// SIMATIC S7-200 project (STEP 7-Micro/WIN), CPU 221 REL 01.10

SYMBOL_TABLE USER1
bezczynnosc_do_za_gorac M1.7     // w彻cz wiatrak
bezczynnosc_do_za_zimno M1.6     // w彻cz grzanie
ANDwb            M1.5     // wy彻czenie wiatraka
ANDgb            M1.4     // wy彻czenie grza砶i
RSwentylator     M1.3
RSgrzalka        M1.2
RSbezczynnosc    M1.1
ANDgrzalka       M0.6
bezczynnosc      M0.5
ANDwentylator    M0.7
T_z_sub_h        VW130
T_z_add_h        VW120
h                VW110
T_ge_T_z         M0.2
T_z_ge_T         M0.1
h_count          C1
T_z              VW100
T_z_count        C0
T                AIW8
END_SYMBOL_TABLE

ORGANIZATION_BLOCK MAIN:OB1
TITLE=PROGRAM COMMENTS
BEGIN
Network 1 // Network Title
// Counter temp zadana
LD     I0.0
LD     I0.1
LD     SM0.1
CTUD   T_z_count:C0, 0
Network 2
// Temperatura zadana
// (network saved uncompiled; FBD cells follow)
// row 0: c1 [ADD_I ]
// row 1: c1 [ EN:=SM0.0, IN1:=T_z_count:C0, IN2:=+220, ENO=>V?0, OUT=>T_z:VW100]
// row 2: c1 [box]
// row 3: c1 [box]
Network 3
// Counter histereza
LD     I0.2
LD     I0.3
LD     SM0.1
CTUD   h_count:C1, 0
Network 4
// Histereza
// (network saved uncompiled; FBD cells follow)
// row 0: c1 [ADD_I ]
// row 1: c1 [ EN:=SM0.0, IN1:=h_count:C1, IN2:=+6, ENO=>V?0, OUT=>h:VW110]
// row 2: c1 [box]
// row 3: c1 [box]
Network 5
// Temperetura zadana + histereza
// (network saved uncompiled; FBD cells follow)
// row 0: c1 [ADD_I ]
// row 1: c1 [ EN:=SM0.0, IN1:=T_z:VW100, IN2:=h:VW110, ENO=>V?0, OUT=>T_z_add_h:VW120]
// row 2: c1 [box]
// row 3: c1 [box]
Network 6
// Tempreatura zadana - histereza
// (network saved uncompiled; FBD cells follow)
// row 0: c1 [SUB_I ]
// row 1: c1 [ EN:=SM0.0, IN1:=T_z:VW100, IN2:=h:VW110, ENO=>V?0, OUT=>T_z_sub_h:VW130]
// row 2: c1 [box]
// row 3: c1 [box]
Network 7 // PID
// (network saved uncompiled; FBD cells follow)
// row 0: c1 [PID0_INIT ]
// row 1: c1 [ EN:=SM0.0, PV_I:=T:AIW8, Setpoint_R:=VD0, Output=>AQW0]
// row 2: c1 [box]
// row 3: c1 [box]
Network 8
// AND grzalka
LDW>   T_z_sub_h:VW130, T:AIW8
A      RSbezczynnosc:M1.1
=      ANDgrzalka:M0.6
Network 9
// AND grzalka -> bezczynnosc
LDW>=  T:AIW8, T_z:VW100
A      RSgrzalka:M1.2
=      ANDgb:M1.4
Network 10
// AND wentylator -> bezczynnosc
LDW<=  T:AIW8, T_z:VW100
A      RSwentylator:M1.3
=      ANDwb:M1.5
Network 11
// (network saved uncompiled; FBD cells follow)
// row 1: c1 [OR SM0.1 ANDgb:M1.4 ]  c2 --  c3 [RS Q0.3 S:=power@row1, R1:=ANDgrzalka:M0.6, OUT=>RSbezczynnosc:M1.1]
// row 2: c1 [box]  c3 [box]
// row 3: c3 [box]
// row 4: c3 [box]
Network 12
// w彻cz grzanie
LD     ANDgrzalka:M0.6
LD     ANDgb:M1.4
NOT
LPS
A      Q0.2
=      Q0.2
LPP
ALD
O      Q0.2
=      Q0.2
=      RSgrzalka:M1.2
END_ORGANIZATION_BLOCK

// SBR1: protected block, not included

// INT1: protected block, not included

// (further data pages could not be read)
